FUNCTION_BLOCK Circuit_Breaker (* Composite Function Block Type *)
  (* Standard: 61499-2 *)
  (* Version 0.0, 12/11/2023, Cheyan, Schneider Electric, template *)
  PACKAGE Main;
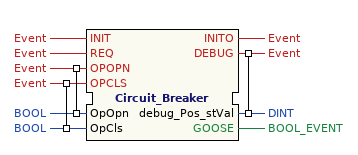
  EVENT_INPUT
    INIT; (* Initialization Request *)
    REQ; (* Normal Execution Request *)
    OPOPN WITH OpOpn;
    OPCLS WITH OpCls;
  END_EVENT
  EVENT_OUTPUT
    INITO; (* Initialization Confirm *)
    DEBUG WITH debug_Pos_stVal;
  END_EVENT
  VAR_INPUT
    OpOpn : BOOL; (* Input event qualifier *)
    OpCls : BOOL;
  END_VAR
  VAR_OUTPUT
    debug_Pos_stVal : DINT;
  END_VAR
  PLUGS
    GOOSE : BOOL_EVENT;
  END_PLUGS
  FBS
    FB1 : XCBR_Logic;
  END_FBS
  EVENT_CONNECTIONS
    INIT TO FB1.INIT;
    REQ TO FB1.REQ;
    FB1.INITO TO INITO;
    FB1.OPERATE_CB TO GOOSE.ACTUATE;
    FB1.DEBUG TO DEBUG;
    OPOPN TO FB1.OPOPN;
    OPCLS TO FB1.OPCLS;
  END_CONNECTIONS
  DATA_CONNECTIONS
    FB1.openCB TO GOOSE.openSwitch;
    FB1.debug_Pos_stVal TO debug_Pos_stVal;
    OpOpn TO FB1.OpOpn;
    OpCls TO FB1.OpCls;
  END_CONNECTIONS
END_FUNCTION_BLOCK
